{attribute 'linkalways'} 
{attribute 'no_explicit_call' := 'This FB is a CLASS and must be accessed using methods or properties'}
{attribute 'enable_dynamic_creation'}
FUNCTION_BLOCK Node_ContainerType_Vector_TcVnVector3_SINT EXTENDS Node
VAR
    out : _GUID;
END_VAR

METHOD PUBLIC  Clone : I_Node
VAR
	pNode : POINTER TO Node_ContainerType_Vector_TcVnVector3_SINT;
END_VAR
pNode := __NEW(Node_ContainerType_Vector_TcVnVector3_SINT);
Clone := pNode^;
END_METHOD

METHOD FB_init : BOOL
VAR_INPUT
	bInitRetains : BOOL; // if TRUE, the retain variables are initialized (warm start / cold start)
	bInCopyCode : BOOL;  // if TRUE, the instance afterwards gets moved into the copy code (online change)
END_VAR
AddOutput('out', out);
END_METHOD

METHOD PROTECTED OnExecute
out.Value := ContainerType_Vector_TcVnVector3_SINT;
END_METHOD

END_FUNCTION_BLOCK

(* stored: Version 1.1.0.1, ProductVersion 3.1.4026.17
   POU Node_ContainerType_Vector_TcVnVector3_SINT: Id {ed55fb75-26aa-0e0a-1317-f5ad742e87aa}, SpecialFunc None
   Folder Constructor: Id {3cab1b2f-c841-0aff-2d1e-0636c69430ec}
   Method Clone: Id {e24b24f7-6279-0d20-1f67-2347e31ff202}
   Method FB_init: Id {7dcd1670-8b16-0ab1-31aa-8b9ff7845001}
   Method OnExecute: Id {c4dab87e-8581-0f9a-2150-5e78e62e8ea0} *)
